TYPE ST_Debounce :
STRUCT
	RawSignal : BOOL;
	DebSignal : BOOL;
END_STRUCT
END_TYPE

(* stored: Version 1.1.0.1
   DUT ST_Debounce: Id {c2874131-500f-0506-1479-a848ecab028b} *)
